// TIA Portal V16 export
// export: Created 2024-09-05T17:39:20.1346803Z, ExportSetting WithDefaults, DisplayName Totally Integrated Automation Portal, DisplayVersion V16 Update 6, DisplayName TIA Portal Version Control Interface, DisplayVersion V16 Update 2, DisplayName TIA Portal Openness, DisplayVersion V16 Update 6, DisplayName STEP 7 Professional, DisplayVersion V16 Update 6, DisplayName STEP 7 Safety, DisplayVersion V16, DisplayName WinCC Advanced, DisplayVersion V16 Update 6
FUNCTION_BLOCK "sq_robot"   // FB42, GRAPH
VERSION : 0.1
// stored: AcknowledgeErrorsRequired true, AutoNumber true, GraphVersion 6.0, InitialValuesAcquisition false, IsIECCheckEnabled false, LanguageInNetworks LAD, LockOperatingMode false, PermanentILProcessingInMANMode false, SetENOAutomatically false, SkipSteps false, UDAEnableTagReadback false, WithAlarmHandling true
   // inherited from GRAPH_BASE
   VAR
      OFF_SQ_BASE : Bool;
   END_VAR
   VAR_INPUT
      OFF_SQ { ExternalWritable := 'False'} : Bool := false;   // Turn sequence off
      INIT_SQ { ExternalWritable := 'False'} : Bool := false;   // Set sequence to initial state
      ACK_EF { ExternalWritable := 'False'} : Bool := false;   // Acknowledge all errors and faults
      S_PREV { ExternalWritable := 'False'} : Bool := false;   // Output previous step in parameter S_NO
      S_NEXT { ExternalWritable := 'False'} : Bool := false;   // Indicate next step in parameter S_NO
      SW_AUTO { ExternalWritable := 'False'} : Bool := false;   // Automatic mode
      SW_TAP { ExternalWritable := 'False'} : Bool := false;   // Semiautomatic/switch with transition
      SW_TOP { ExternalWritable := 'False'} : Bool := false;   // Semiautomatic/ignore transition
      SW_MAN { ExternalWritable := 'False'} : Bool := false;   // Manual mode
      S_SEL { ExternalWritable := 'False'} : Int := 0;   // Select step to be output to S_NO
      S_ON { ExternalWritable := 'False'} : Bool := false;   // Activate step indicated in S_NO
      S_OFF { ExternalWritable := 'False'} : Bool := false;   // Deactivate step indicated S_NO
      T_PUSH { ExternalWritable := 'False'} : Bool := false;   // Enable transition to switch in semi automatic mode
   END_VAR
   VAR_OUTPUT
      S_NO { ExternalWritable := 'False'} : Int := 0;   // Step number
      S_MORE { ExternalWritable := 'False'} : Bool := false;   // More steps are available and can be shown in S_NO
      S_ACTIVE { ExternalWritable := 'False'} : Bool := false;   // Step indicated in S_NO is active
      ERR_FLT { ExternalWritable := 'False'} : Bool := false;   // Interlock or supervision group error
      AUTO_ON { ExternalWritable := 'False'} : Bool := false;   // Automatic mode is active
      TAP_ON { ExternalWritable := 'False'} : Bool := false;   // Semiautomatic mode/step with transition enabled
      TOP_ON { ExternalWritable := 'False'} : Bool := false;   // Semiautomatic mode/ignore transition enabled
      MAN_ON { ExternalWritable := 'False'} : Bool := false;   // Manual mode is active
   END_VAR
   VAR
      dummy : Bool;
      start : Bool;
      base : Bool;
      startMastering : Bool;
      startBraketest : Bool;
      prgNrForManipulatorDropoff : Byte;
   END_VAR
   VAR CONSTANT
      jobHoming : Byte := 1;
      jobCarouselPickup : Byte := 2;
      jobJigDropoff : Byte := 3;
      jobAutoEjectPickup : Byte := 4;
      jobMastering : Byte := 10;
      jobBreaktest : Byte := 11;
      jobManipulatorDropoff1 : Byte := 21;   // top far
      jobManipulatorDropoff2 : Byte := 22;   // top middle
      jobManipulatorDropoff3 : Byte := 23;   // top near
      jobManipulatorDropoff4 : Byte := 24;   // bottom far
      jobManipulatorDropoff5 : Byte := 25;   // bottom middle
      jobManipulatorDropoff6 : Byte := 26;   // bottom near
      jobManipulatorForTesting : Byte := 30;
   END_VAR
   VAR_TEMP   // added for the SCL form of the ladder/FBD networks
      _w1 : Bool;
      _w2 : Bool;
   END_VAR
BEGIN
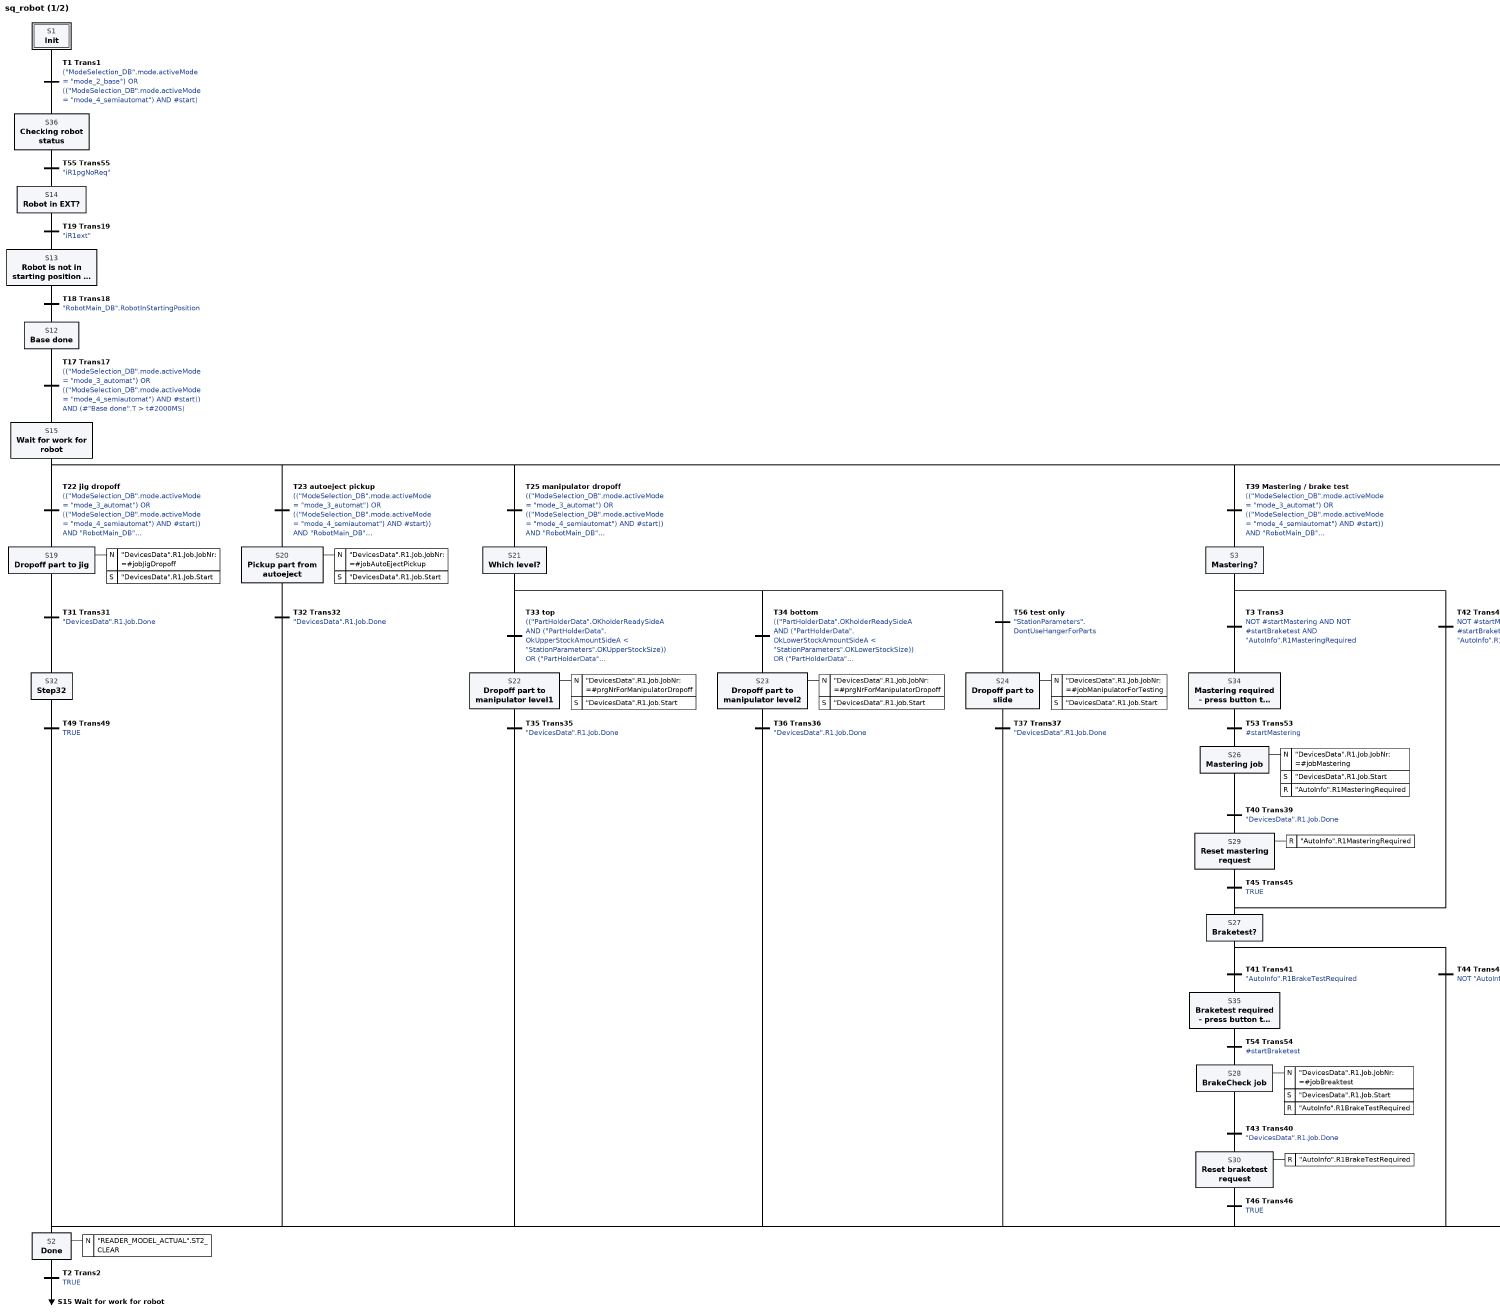
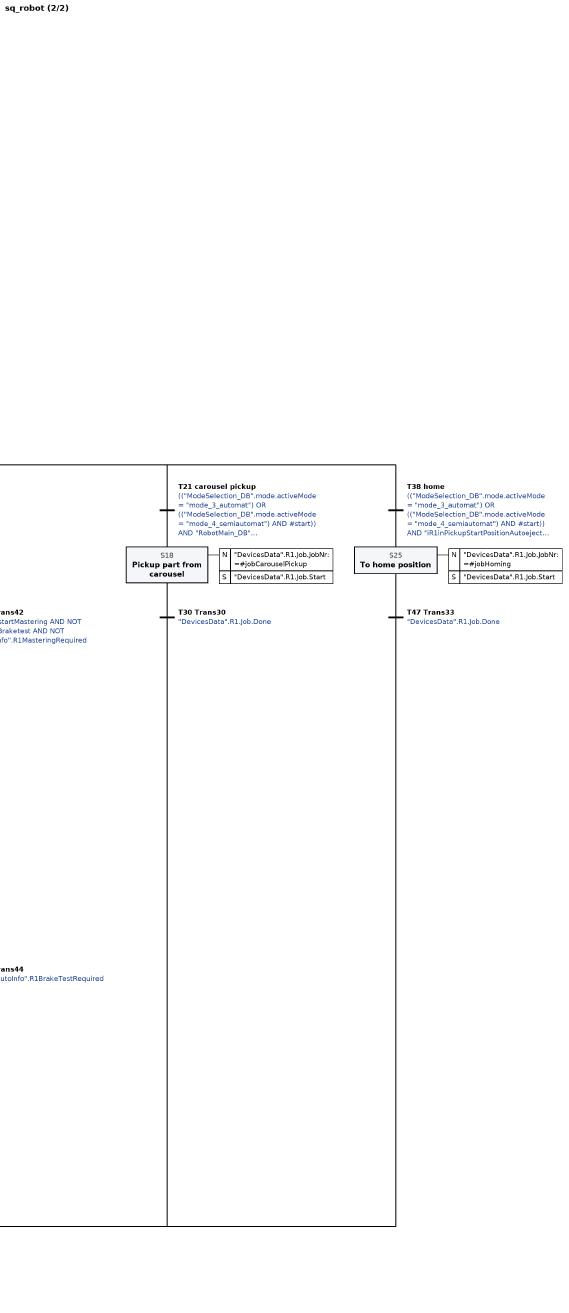
   // permanent pre-instructions
   NETWORK 1
   TITLE = prg for top level
      #_w1 := #"Dropoff part to manipulator level1".S1 AND "PartHolderData".OKholderReadySideA AND NOT "PartHolderData".OKholderReadySideB;
      IF #_w1 AND ("PartHolderData".OkUpperStockAmountSideA = 0) THEN
          #prgNrForManipulatorDropoff := #jobManipulatorDropoff1;
      END_IF;
      IF #_w1 AND ("PartHolderData".OkUpperStockAmountSideA = 1) THEN
          #prgNrForManipulatorDropoff := #jobManipulatorDropoff2;
      END_IF;
      IF #_w1 AND ("PartHolderData".OkUpperStockAmountSideA = 2) THEN
          #prgNrForManipulatorDropoff := #jobManipulatorDropoff3;
      END_IF;
      #_w2 := #"Dropoff part to manipulator level1".S1 AND NOT "PartHolderData".OKholderReadySideA AND "PartHolderData".OKholderReadySideB;
      IF #_w2 AND ("PartHolderData".OkUpperStockAmountSideB = 0) THEN
          #prgNrForManipulatorDropoff := #jobManipulatorDropoff1;
      END_IF;
      IF #_w2 AND ("PartHolderData".OkUpperStockAmountSideB = 1) THEN
          #prgNrForManipulatorDropoff := #jobManipulatorDropoff2;
      END_IF;
      IF #_w2 AND ("PartHolderData".OkUpperStockAmountSideB = 2) THEN
          #prgNrForManipulatorDropoff := #jobManipulatorDropoff3;
      END_IF;
   NETWORK 2
   TITLE = prg for bottom level
      #_w1 := #"Dropoff part to manipulator level2".S1 AND "PartHolderData".OKholderReadySideA AND NOT "PartHolderData".OKholderReadySideB;
      IF #_w1 AND ("PartHolderData".OkLowerStockAmountSideA = 0) THEN
          #prgNrForManipulatorDropoff := #jobManipulatorDropoff4;
      END_IF;
      IF #_w1 AND ("PartHolderData".OkLowerStockAmountSideA = 1) THEN
          #prgNrForManipulatorDropoff := #jobManipulatorDropoff5;
      END_IF;
      IF #_w1 AND ("PartHolderData".OkLowerStockAmountSideA = 2) THEN
          #prgNrForManipulatorDropoff := #jobManipulatorDropoff6;
      END_IF;
      #_w2 := #"Dropoff part to manipulator level2".S1 AND NOT "PartHolderData".OKholderReadySideA AND "PartHolderData".OKholderReadySideB;
      IF #_w2 AND ("PartHolderData".OkLowerStockAmountSideB = 0) THEN
          #prgNrForManipulatorDropoff := #jobManipulatorDropoff4;
      END_IF;
      IF #_w2 AND ("PartHolderData".OkLowerStockAmountSideB = 1) THEN
          #prgNrForManipulatorDropoff := #jobManipulatorDropoff5;
      END_IF;
      IF #_w2 AND ("PartHolderData".OkLowerStockAmountSideB = 2) THEN
          #prgNrForManipulatorDropoff := #jobManipulatorDropoff6;
      END_IF;
   NETWORK 3
      #base := "RobotMain_DB".RobotInStartingPosition AND "iR1ext";
   NETWORK 4
   TITLE = job start init
      "DevicesData".R1.Job.Start := FALSE;
   NETWORK 5
      "qR1_ST3free" := "sq_fitting_station_st3".base;

   // sequencer 1
   INITIAL_STEP Init:   // S1, max time T#10S, warning time T#7S
   END_STEP
   TRANSITION Trans1 FROM Init TO "Checking robot status"   // T1
      := ("ModeSelection_DB".mode.activeMode = "mode_2_base") OR (("ModeSelection_DB".mode.activeMode = "mode_4_semiautomat") AND #start);
   END_TRANSITION
   STEP Done:   // S2, max time T#10S, warning time T#7S
              N    "READER_MODEL_ACTUAL".ST2_CLEAR
   END_STEP
   TRANSITION Trans2 FROM Done TO "Wait for work for robot"   // T2, jump
      := TRUE;
   END_TRANSITION
   STEP "Base done":   // S12, max time T#10S, warning time T#7S
   END_STEP
   TRANSITION Trans17 FROM "Base done" TO "Wait for work for robot"   // T17
      := (("ModeSelection_DB".mode.activeMode = "mode_3_automat") OR (("ModeSelection_DB".mode.activeMode = "mode_4_semiautomat") AND #start)) AND (#"Base done".T > t#2000MS);
   END_TRANSITION
   STEP "Robot is not in starting position - move it to home manualy":   // S13, max time T#1S, warning time T#7S
      supervision V := #"Robot is not in starting position - move it to home manualy".T > #"Robot is not in starting position - move it to home manualy".T_MAX;
   END_STEP
   TRANSITION Trans18 FROM "Robot is not in starting position - move it to home manualy" TO "Base done"   // T18
      := "RobotMain_DB".RobotInStartingPosition;
   END_TRANSITION
   STEP "Robot in EXT?":   // S14, max time T#10S, warning time T#7S
      supervision V := #"Robot in EXT?".T > #"Robot in EXT?".T_MAX;
   END_STEP
   TRANSITION Trans19 FROM "Robot in EXT?" TO "Robot is not in starting position - move it to home manualy"   // T19
      := "iR1ext";
   END_TRANSITION
   STEP "Wait for work for robot":   // S15, max time T#10S, warning time T#7S
   END_STEP
   TRANSITION "jig dropoff" FROM "Wait for work for robot" TO "Dropoff part to jig"   // T22
      := (("ModeSelection_DB".mode.activeMode = "mode_3_automat") OR (("ModeSelection_DB".mode.activeMode = "mode_4_semiautomat") AND #start)) AND "RobotMain_DB".RobotInStartingPosition AND "sq_fitting_station_st3"."Waiting for the part to be inserted".X AND "DevicesData"."TA1-3MA".data.zones.outOfST3zone AND NOT "AutoPositions".St3_Fitting.PartPresent AND NOT "i3partPresent" AND "AutoPositions".R1_Gripper.PartPresent AND "iR1tubePresentFront" AND "iR1tubePresentRear" AND NOT "AutoPositions".R1_Gripper.StFinished[3] AND NOT "AutoPositions".R1_Gripper.PartNOK AND "sq_fitting_station_st3".base;
   END_TRANSITION
   TRANSITION "autoeject pickup" FROM "Wait for work for robot" TO "Pickup part from autoeject"   // T23
      := (("ModeSelection_DB".mode.activeMode = "mode_3_automat") OR (("ModeSelection_DB".mode.activeMode = "mode_4_semiautomat") AND #start)) AND "RobotMain_DB".RobotInStartingPosition AND "DevicesData"."TA1-3MA".data.zones.outOfOKposZone AND ((NOT "AutoInfo".EndProduction AND "AutoPositions".St3_Fitting.PartPresent) OR "AutoInfo".EndProduction) AND ("i4partPresent" OR "StationParameters".GhostMode) AND NOT "AutoPositions".R1_Gripper.PartPresent AND NOT "iR1tubePresentFront" AND NOT "iR1tubePresentRear" AND "AutoPositions".St4_OKposition.PartPresent;
   END_TRANSITION
   TRANSITION "manipulator dropoff" FROM "Wait for work for robot" TO "Which level?"   // T25
      := (("ModeSelection_DB".mode.activeMode = "mode_3_automat") OR (("ModeSelection_DB".mode.activeMode = "mode_4_semiautomat") AND #start)) AND "RobotMain_DB".RobotInStartingPosition AND (("PartHolderData".OKholderReadySideA AND (("PartHolderData".OkLowerStockAmountSideA < "StationParameters".OKLowerStockSize) OR ("PartHolderData".OkUpperStockAmountSideA < "StationParameters".OKUpperStockSize))) OR ("PartHolderData".OKholderReadySideB AND (("PartHolderData".OkLowerStockAmountSideB < "StationParameters".OKLowerStockSize) OR ("PartHolderData".OkUpperStockAmountSideB < "StationParameters".OKUpperStockSize)))) AND "AutoPositions".R1_Gripper.PartPresent AND "iR1tubePresentFront" AND "iR1tubePresentRear" AND "AutoPositions".R1_Gripper.StFinished[3] AND NOT "AutoPositions".R1_Gripper.PartNOK;
   END_TRANSITION
   TRANSITION "Mastering / brake test" FROM "Wait for work for robot" TO "Mastering?"   // T39
      := (("ModeSelection_DB".mode.activeMode = "mode_3_automat") OR (("ModeSelection_DB".mode.activeMode = "mode_4_semiautomat") AND #start)) AND "RobotMain_DB".RobotInStartingPosition AND "DevicesData"."TA1-3MA".data.zones.outOfST3zone AND NOT "AutoPositions".R1_Gripper.PartPresent AND NOT "iR1tubePresentFront" AND NOT "iR1tubePresentRear" AND ("AutoInfo".R1MasteringRequired OR "AutoInfo".R1BrakeTestRequired);
   END_TRANSITION
   TRANSITION "carousel pickup" FROM "Wait for work for robot" TO "Pickup part from carousel"   // T21
      := (("ModeSelection_DB".mode.activeMode = "mode_3_automat") OR (("ModeSelection_DB".mode.activeMode = "mode_4_semiautomat") AND #start)) AND "RobotMain_DB".RobotInStartingPosition AND "sq_carousel_unloading_st2"."Wait for robot to remove part".X AND "AutoPositions".St2_Table2.PartPresent AND (NOT "AutoPositions".St3_Fitting.PartPresent OR NOT "AutoPositions".St4_OKposition.PartPresent) AND NOT "AutoPositions".St2_Table2.PartNOK AND NOT "AutoPositions".R1_Gripper.PartPresent AND NOT "iR1tubePresentFront" AND NOT "iR1tubePresentRear" AND "iTableInPosition" AND "iTurnTableIndexerInPosition";
   END_TRANSITION
   TRANSITION home FROM "Wait for work for robot" TO "To home position"   // T38
      := (("ModeSelection_DB".mode.activeMode = "mode_3_automat") OR (("ModeSelection_DB".mode.activeMode = "mode_4_semiautomat") AND #start)) AND "iR1inPickupStartPositionAutoeject" AND "AutoInfo".EndProduction AND NOT "AutoPositions".St2_Table2.PartPresent AND "AutoPositions".St3_Fitting.PartPresent AND "i3partPresent" AND NOT "AutoPositions".St4_OKposition.PartPresent AND NOT "i4partPresent";
   END_TRANSITION
   STEP "Mastering job":   // S26, max time T#50S, warning time T#7S
      supervision V := #"Mastering job".T > #"Mastering job".T_MAX;
              N    "DevicesData".R1.Job.JobNr:=#jobMastering
              S    "DevicesData".R1.Job.Start
              R    "AutoInfo".R1MasteringRequired
   END_STEP
   TRANSITION Trans39 FROM "Mastering job" TO "Reset mastering request"   // T40
      := "DevicesData".R1.Job.Done;
   END_TRANSITION
   STEP "Dropoff part to jig":   // S19, max time T#30S, warning time T#7S
      supervision V := #"Dropoff part to jig".T > #"Dropoff part to jig".T_MAX;
              N    "DevicesData".R1.Job.JobNr:=#jobJigDropoff
              S    "DevicesData".R1.Job.Start
   END_STEP
   TRANSITION Trans31 FROM "Dropoff part to jig" TO Step32   // T31
      := "DevicesData".R1.Job.Done;
   END_TRANSITION
   STEP "Pickup part from autoeject":   // S20, max time T#30S, warning time T#7S
      supervision V := #"Pickup part from autoeject".T > #"Pickup part from autoeject".T_MAX;
              N    "DevicesData".R1.Job.JobNr:=#jobAutoEjectPickup
              S    "DevicesData".R1.Job.Start
   END_STEP
   TRANSITION Trans32 FROM "Pickup part from autoeject" TO Done   // T32
      := "DevicesData".R1.Job.Done;
   END_TRANSITION
   STEP "Which level?":   // S21, max time T#10S, warning time T#7S
   END_STEP
   TRANSITION top FROM "Which level?" TO "Dropoff part to manipulator level1"   // T33
      := (("PartHolderData".OKholderReadySideA AND ("PartHolderData".OkUpperStockAmountSideA < "StationParameters".OKUpperStockSize)) OR ("PartHolderData".OKholderReadySideB AND ("PartHolderData".OkUpperStockAmountSideB < "StationParameters".OKUpperStockSize))) AND NOT "StationParameters".DontUseHangerForParts;
   END_TRANSITION
   TRANSITION bottom FROM "Which level?" TO "Dropoff part to manipulator level2"   // T34
      := (("PartHolderData".OKholderReadySideA AND ("PartHolderData".OkLowerStockAmountSideA < "StationParameters".OKLowerStockSize)) OR ("PartHolderData".OKholderReadySideB AND ("PartHolderData".OkLowerStockAmountSideB < "StationParameters".OKLowerStockSize))) AND NOT "StationParameters".DontUseHangerForParts;
   END_TRANSITION
   TRANSITION "test only" FROM "Which level?" TO "Dropoff part to slide"   // T56
      := "StationParameters".DontUseHangerForParts;
   END_TRANSITION
   STEP "Dropoff part to manipulator level1":   // S22, max time T#30S, warning time T#7S
      supervision V := (#"Dropoff part to manipulator level1".T > #"Dropoff part to manipulator level1".T_MAX) AND (#"Dropoff part to manipulator level1".T > T#60S);
              N    "DevicesData".R1.Job.JobNr:=#prgNrForManipulatorDropoff
              S    "DevicesData".R1.Job.Start
   END_STEP
   TRANSITION Trans35 FROM "Dropoff part to manipulator level1" TO Done   // T35
      := "DevicesData".R1.Job.Done;
   END_TRANSITION
   STEP "Dropoff part to manipulator level2":   // S23, max time T#30S, warning time T#7S
      supervision V := #"Dropoff part to manipulator level2".T > #"Dropoff part to manipulator level2".T_MAX;
              N    "DevicesData".R1.Job.JobNr:=#prgNrForManipulatorDropoff
              S    "DevicesData".R1.Job.Start
   END_STEP
   TRANSITION Trans36 FROM "Dropoff part to manipulator level2" TO Done   // T36
      := "DevicesData".R1.Job.Done;
   END_TRANSITION
   STEP "Mastering?":   // S3, max time T#10S, warning time T#7S
   END_STEP
   TRANSITION Trans3 FROM "Mastering?" TO "Mastering required - press button to start"   // T3
      := NOT #startMastering AND NOT #startBraketest AND "AutoInfo".R1MasteringRequired;
   END_TRANSITION
   TRANSITION Trans42 FROM "Mastering?" TO "Braketest?"   // T42
      := NOT #startMastering AND NOT #startBraketest AND NOT "AutoInfo".R1MasteringRequired;
   END_TRANSITION
   STEP "Pickup part from carousel":   // S18, max time T#30S, warning time T#7S
      supervision V := #"Pickup part from carousel".T > #"Pickup part from carousel".T_MAX;
              N    "DevicesData".R1.Job.JobNr:=#jobCarouselPickup
              S    "DevicesData".R1.Job.Start
   END_STEP
   TRANSITION Trans30 FROM "Pickup part from carousel" TO Done   // T30
      := "DevicesData".R1.Job.Done;
   END_TRANSITION
   STEP "Braketest?":   // S27, max time T#10S, warning time T#7S
   END_STEP
   TRANSITION Trans41 FROM "Braketest?" TO "Braketest required - press button to start"   // T41
      := "AutoInfo".R1BrakeTestRequired;
   END_TRANSITION
   TRANSITION Trans44 FROM "Braketest?" TO Done   // T44
      := NOT "AutoInfo".R1BrakeTestRequired;
   END_TRANSITION
   STEP "BrakeCheck job":   // S28, max time T#60S, warning time T#7S
      supervision V := #"BrakeCheck job".T > #"BrakeCheck job".T_MAX;
              N    "DevicesData".R1.Job.JobNr:=#jobBreaktest
              S    "DevicesData".R1.Job.Start
              R    "AutoInfo".R1BrakeTestRequired
   END_STEP
   TRANSITION Trans40 FROM "BrakeCheck job" TO "Reset braketest request"   // T43
      := "DevicesData".R1.Job.Done;
   END_TRANSITION
   STEP "Reset mastering request":   // S29, max time T#10S, warning time T#7S
              R    "AutoInfo".R1MasteringRequired
   END_STEP
   TRANSITION Trans45 FROM "Reset mastering request" TO "Braketest?"   // T45
      := TRUE;
   END_TRANSITION
   STEP "Reset braketest request":   // S30, max time T#10S, warning time T#7S
              R    "AutoInfo".R1BrakeTestRequired
   END_STEP
   TRANSITION Trans46 FROM "Reset braketest request" TO Done   // T46
      := TRUE;
   END_TRANSITION
   STEP "Mastering required - press button to start":   // S34, max time T#10S, warning time T#7S
   END_STEP
   TRANSITION Trans53 FROM "Mastering required - press button to start" TO "Mastering job"   // T53
      := #startMastering;
   END_TRANSITION
   STEP "Braketest required - press button to start":   // S35, max time T#10S, warning time T#7S
   END_STEP
   TRANSITION Trans54 FROM "Braketest required - press button to start" TO "BrakeCheck job"   // T54
      := #startBraketest;
   END_TRANSITION
   STEP "Checking robot status":   // S36, max time T#10S, warning time T#7S
   END_STEP
   TRANSITION Trans55 FROM "Checking robot status" TO "Robot in EXT?"   // T55
      := "iR1pgNoReq";
   END_TRANSITION
   STEP "Dropoff part to slide":   // S24, max time T#40S, warning time T#7S
      supervision V := #"Dropoff part to slide".T > #"Dropoff part to slide".T_MAX;
              N    "DevicesData".R1.Job.JobNr:=#jobManipulatorForTesting
              S    "DevicesData".R1.Job.Start
   END_STEP
   TRANSITION Trans37 FROM "Dropoff part to slide" TO Done   // T37
      := "DevicesData".R1.Job.Done;
   END_TRANSITION
   STEP "To home position":   // S25, max time T#10S, warning time T#7S
      supervision V := #"To home position".T > #"To home position".T_MAX;
              N    "DevicesData".R1.Job.JobNr:=#jobHoming
              S    "DevicesData".R1.Job.Start
   END_STEP
   TRANSITION Trans33 FROM "To home position" TO Done   // T47
      := "DevicesData".R1.Job.Done;
   END_TRANSITION
   STEP Step32:   // S32, max time T#10S, warning time T#7S
   END_STEP
   TRANSITION Trans49 FROM Step32 TO Done   // T49
      := TRUE;
   END_TRANSITION

   // permanent post-instructions
   NETWORK 1
      IF #startMastering THEN #startMastering := FALSE; END_IF;
      IF #startBraketest THEN #startBraketest := FALSE; END_IF;
END_FUNCTION_BLOCK
